TYPE LogEvent :
STRUCT
	(*~
	<docu>
		<summary>
			Time when the message was posted.
		</summary>				
	</docu>	
~*)
	{attribute clr [ReadOnly()]}
	TimeStamp : DT;
(*~
	<docu>
		<summary>
			Text of the message.
		</summary>				
	</docu>	
~*)
	{attribute clr [ReadOnly()]}		
	Text : STRING(255);
(*~
	<docu>
		<summary>
			Identity of the TcoObject that posted this message. 
		</summary>				
	</docu>	
~*)
	{attribute clr [ReadOnly()]}	
	Identity : ULINT;	
(*~
	<docu>
		<summary>
			Message category of this message. See <see cref="eMessageCategory"/> for detailed informations. 
		</summary>				
	</docu>	
~*)
	LogLevel : LogLevel;
(*~
	<docu>
		<summary>
			Context cycle in which the message was posted.
		</summary>				
	</docu>	
~*)
	{attribute clr [ReadOnly()]}
	Cycle : ULINT;
	
(*~
	<docu>
		<summary>
			Count of messages of the object in the current cycle.
		</summary>				
	</docu>	
~*)
	{attribute clr [ReadOnly()]}
	PerCycleCount : BYTE;
END_STRUCT
END_TYPE

(* stored: Version 1.1.0.1, ProductVersion 3.1.4024.9
   DUT LogEvent: Id {765edee2-54fb-0d37-17d3-bf8a2543f15e} *)
